FUNCTION_BLOCK FB_Vereinzelung 
VAR_INPUT
	//Steuervariablen
	benable : BOOL;
	bexecute : BOOL;
	// Hardware Eingänge
	bsensor1 : BOOL; //Flasche in der Kammer 
	bsensor2 : BOOL; //Flasche inm Rohr 
	bsensor3 : BOOL; //Flasche auf Kopf
	bsensor4 : BOOL; //Flasche am Förderband
	
END_VAR
VAR_OUTPUT
	//Hardwareausgänge 
	bgate1 : BOOL;
	bgate2 : BOOL;
	//Steuervariable 
	estate : eBetriebszustand;
END_VAR
VAR
	nstate : INT := 100;
	fbTon : Ton;
END_VAR

fbTon(IN:= , PT:=T#1S , Q=> , ET=> );

CASE nstate OF 
	100:
	eState :=eBetriebszustand.off;
	
	IF bsensor1 AND benable THEN 
		nstate := 21;//Ready
	ELSIF benable THEN
		nstate := 0; //Init		
	END_IF
	
	0: // Kammer ist leer 
	estate := eBetriebszustand.init;
	bgate1 := FALSE;
	bgate2 := FALSE;
	
	IF bsensor2 AND NOT bsensor3 THEN
		nstate := 1; //Schleuße Oben öffnen
	END_IF
	
	1: // Schleuße oben öffnen
	estate := eBetriebszustand.init;
	bgate1 := TRUE;
	bgate2 := FALSE;
	
	IF bsensor1 THEN
		nstate := 2; //Schleuße oben schließen
	END_IF
	
	2: //Schleuße oben schließen
	estate := eBetriebszustand.init;
	bgate1 := FALSE;
	bgate2 := FALSE;
	fbTon.In := TRUE;
	
	IF fbTon.Q THEN
		nstate := 21; //ready
		fbTon.IN := FALSE;
	END_IF
	
	21: //ready
	estate:= eBetriebszustand.ready;
	bgate1:= FALSE;
	bgate2:= FALSE;
	
	
	IF bexecute THEN
		nstate := 3; //Schleuße unten öffnen
	END_IF
	
	3: //Schleuße unten öffnen
	estate:= eBetriebszustand.production;
	bgate1:= FALSE;
	bgate2:= TRUE;
	
	IF bsensor4 THEN
		nstate := 4; //Schleuße unten schließen
	END_IF
	
	4: //Schleuße unten schließen
	estate:= eBetriebszustand.production;
	bgate1:= FALSE;
	bgate2:= FALSE;
	fbTon.IN:= TRUE;
	
	IF fbTon.Q THEN
		nstate := 41; //done
		fbTon.IN := FALSE;
	END_IF	
	
	41: //Done
	estate:= eBetriebszustand.done;
	bgate1:= FALSE;
	bgate2:= FALSE;
	
	IF NOT bexecute THEN
		nstate:= 0; //Kammer leer
	END_IF
	
END_CASE

END_FUNCTION_BLOCK

(* stored: Version 1.1.0.1, ProductVersion 3.1.4024.15
   POU FB_Vereinzelung: Id {f24c2d52-802e-40a8-8120-6923e0b02308}, SpecialFunc None *)
